// TwinCAT 3 PLC project Untitled1
// ProgramVersion: 3.1.4022.3
// libraries:
//   Tc2_Standard, * (Beckhoff Automation GmbH)
//   Tc2_System, * (Beckhoff Automation GmbH)
//   Tc3_Module, * (Beckhoff Automation GmbH)
// project tree:
//   GVLs/ GVL.TcGVL
//   / PlcTask.TcTTO
//   POUs/ Integrator.TcPOU, MAIN.TcPOU
// real-time tasks:
//   TASK PlcTask: cycle T#10ms, priority 20, ADS port 350

CONFIGURATION Untitled1
    RESOURCE PLC ON TwinCAT3
        TASK PlcTask(INTERVAL := T#10ms, PRIORITY := 20);
        PROGRAM MAIN WITH PlcTask : MAIN;
    END_RESOURCE
END_CONFIGURATION

// ---- GVLs/GVL.TcGVL
{attribute 'qualified_only'}
VAR_GLOBAL
	t_global	:	REAL;
	t_cycle		:	REAL;
END_VAR

// ---- POUs/MAIN.TcPOU
PROGRAM MAIN
VAR
	

END_VAR

END_PROGRAM

// ---- POUs/Integrator.TcPOU
FUNCTION_BLOCK Integrator
VAR_INPUT
	e_k		:	REAL;
END_VAR
VAR_OUTPUT
	u_k		:	REAL;
END_VAR
VAR
	u_k_1	:	REAL;
	e_k_1	:	REAL;
	T		:	REAL	:=	0;
	T_leave	:	REAL	:=	0;
	
END_VAR


IF	GVL.t_global		=	0	THEN
	T:= GVL.t_cycle 	
END_IF

END_FUNCTION_BLOCK
